(* Logix 5000 project; controller Machine_Maintenance_Lab2 vendor 1 type 14 code 155 rev 36.11; software revision 36.00 *)

TASK MainTask (continuous, watchdog 500 ms) : MainProgram

MODULES
   Local : vendor 1 type 14 code 155 (PointIO 0, rev 36.11)
      Discrete_IO : Embedded (PointIO 1, rev 36.11, Output RPI 20 ms)
END_MODULES

PROGRAM MainProgram   (* main routine MainRoutine *)
VAR
   counter : COUNTER := (PRE := 5);
   i_GreenPB : ALIAS FOR Local:1:I.Data.0;
   i_Turnkey : ALIAS FOR Local:1:I.Data.2;
   o_GreenPBLight : ALIAS FOR Local:1:O.Data.0;
   o_RedPBLight : ALIAS FOR Local:1:O.Data.1;
   timer : TIMER := (PRE := 5000);
END_VAR

ROUTINE MainRoutine   (* ladder *)
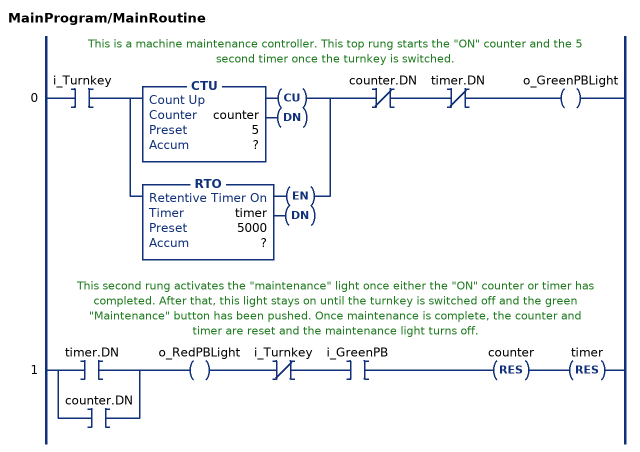
   // This is a machine maintenance controller. This top rung starts the "ON" counter and the 5 second timer once the turnkey is switched.
   0: XIC(i_Turnkey)[CTU(counter,?,?) ,RTO(timer,?,?) ]XIO(counter.DN)XIO(timer.DN)OTE(o_GreenPBLight);
   // This second rung activates the "maintenance" light once either the "ON" counter or timer has completed. After that, this light stays on until the turnkey is switched off and the green "Maintenance" button has been pushed. Once maintenance is complete, the counter and timer are reset and the maintenance light turns off.
   1: [XIC(timer.DN) ,XIC(counter.DN) ]OTE(o_RedPBLight)XIO(i_Turnkey)XIC(i_GreenPB)RES(counter)RES(timer);
END_ROUTINE
END_PROGRAM
